// TIA Portal project "Hardware" (V14)

(* hardware
DEVICE "ET 200S-Station_1"  ET 200S station
   slot 0: "Baugruppenträger_0"  Rail
   slot 2: "PLC_1"  IM151-8 CPU  6ES7 151-8AB00-0AB0  V2.7
      slot 1: "PROFINET-Schnittstelle_1"  PN-IO
         slot 1: "Port_1"  Port
         slot 2: "Port_2"  Port
         slot 3: "Port_3"  Port
   slot 4: "PM-E 24VDC_1"  PM-E 24VDC  6ES7 138-4CA01-0AA0
   slot 5: "4AI x I 2WIRE ST_1"  4AI x I 2WIRE ST  6ES7 134-4GD00-0AB0
   slot 6: "2AO x U ST_1"  2AO x U ST  6ES7 135-4FB01-0AB0
   slot 7: "8DI x 24VDC_1"  8DI x 24VDC  6ES7 131-4BF00-0AA0
   slot 8: "8DI x 24VDC_2"  8DI x 24VDC  6ES7 131-4BF00-0AA0
   slot 9: "8DI x 24VDC_3"  8DI x 24VDC  6ES7 131-4BF00-0AA0
   slot 10: "8DI x 24VDC_4"  8DI x 24VDC  6ES7 131-4BF00-0AA0
   slot 11: "8DO x 24VDC / 0.5A_1"  8DO x 24VDC / 0.5A  6ES7 132-4BF00-0AA0
   slot 12: "8DO x 24VDC / 0.5A_2"  8DO x 24VDC / 0.5A  6ES7 132-4BF00-0AA0
   slot 13: "8DO x 24VDC / 0.5A_3"  8DO x 24VDC / 0.5A  6ES7 132-4BF00-0AA0
   slot 14: "8DO x 24VDC / 0.5A_4"  8DO x 24VDC / 0.5A  6ES7 132-4BF00-0AA0
DEVICE "HMI_1"  TP 177B 6'' PN/DP
   slot 0: "TP 177B 6'' PN/DP"  TP 177B 6'' PN/DP  6AV6 642-0BA01-1AX1  11.0.2.0
   slot 1: "HMI_RT_1"  TP 177B 6'' PN/DP  6AV6 642-0BA01-1AX1  11.0.2.0
   slot 5: "HMI_1.IE_CP_1"  PROFINET Interface  11.0.0.0
      slot 1: "PROFINET Schnittstelle_1"  PROFINET Interface
         slot 1: "Port_1"  Port
   slot 7: "HMI_1.MPI/DP_CP_1"  MPI/DP Interface  11.0.0.0
*)

// ===== PLC "PLC_1"  IM151-8 CPU =====

DATA_BLOCK "DB1"   // DB1
{ S7_Optimized_Access := 'FALSE' }
VERSION : 0.1
   VAR
      Static_0 : Int := 0;
      Static_1 : DInt := 0;
      Static_2 : Real := -1.0;
      Static_3 : Real := -1.0;
      Static_4 : Bool := FALSE;
   END_VAR
BEGIN
END_DATA_BLOCK

DATA_BLOCK "DB2"   // DB2
{ S7_Optimized_Access := 'FALSE' }
VERSION : 0.1
   VAR
      Static_0 : Int := 0;
      Static_1 : Array[0..2, 0..9] of Real;
      Static_2 : Real := 50.0;
      Static_3 : Real := 30.0;
      Static_4 : Real := 20.0;
      Static_5 : Bool := FALSE;
   END_VAR
BEGIN
   Static_1[0,0] := 50.0;
   Static_1[0,1] := 0.0;
   Static_1[0,2] := 0.0;
   Static_1[0,3] := 0.0;
   Static_1[0,4] := 0.0;
   Static_1[0,5] := 0.0;
   Static_1[0,6] := 0.0;
   Static_1[0,7] := 0.0;
   Static_1[0,8] := 0.0;
   Static_1[0,9] := 0.0;
   Static_1[1,0] := 30.0;
   Static_1[1,1] := 0.0;
   Static_1[1,2] := 0.0;
   Static_1[1,3] := 0.0;
   Static_1[1,4] := 0.0;
   Static_1[1,5] := 0.0;
   Static_1[1,6] := 0.0;
   Static_1[1,7] := 0.0;
   Static_1[1,8] := 0.0;
   Static_1[1,9] := 0.0;
   Static_1[2,0] := 20.0;
   Static_1[2,1] := 0.0;
   Static_1[2,2] := 0.0;
   Static_1[2,3] := 0.0;
   Static_1[2,4] := 0.0;
   Static_1[2,5] := 0.0;
   Static_1[2,6] := 0.0;
   Static_1[2,7] := 0.0;
   Static_1[2,8] := 0.0;
   Static_1[2,9] := 0.0;
END_DATA_BLOCK

DATA_BLOCK "DB3"   // DB3
{ S7_Optimized_Access := 'FALSE' }
VERSION : 0.1
   VAR
      Static_0 : Int := 0;
      Static_1 : Int := 0;
      Static_2 : Int := 0;
   END_VAR
BEGIN
END_DATA_BLOCK

DATA_BLOCK "DB100"   // DB100
{ S7_Optimized_Access := 'FALSE' }
VERSION : 0.1
   VAR
      Static_0 : Real := 0.0;
      Static_1 : Real := 0.0;
      Static_2 : Real := 0.0;
   END_VAR
BEGIN
END_DATA_BLOCK

DATA_BLOCK "DB101"   // DB101
{ S7_Optimized_Access := 'FALSE' }
VERSION : 0.1
   VAR
      Static_0 : Int := 0;
   END_VAR
BEGIN
END_DATA_BLOCK

FUNCTION "FC1" : Real   // FC1, FBD
{ S7_Optimized_Access := 'FALSE' }
VERSION : 0.1
   VAR_INPUT
      Input_0 : Int;
      Input_1 : DInt;
   END_VAR
   VAR_TEMP
      Temp_0 : DInt;
      Temp_1 : DInt;
      Temp_2 : DInt;
      Temp_3 : Real;
      Temp_4 : Real;
      Temp_5 : Real;
   END_VAR
BEGIN

REGION Network 1
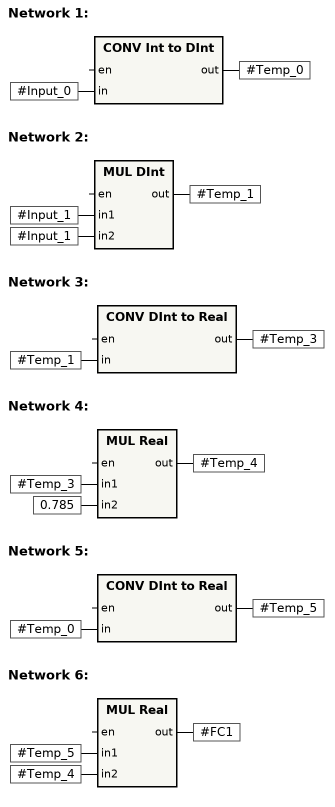
   #Temp_0 := INT_TO_DINT(#Input_0);
END_REGION

REGION Network 2
   #Temp_1 := #Input_1 * #Input_1;
END_REGION

REGION Network 3
   #Temp_3 := DINT_TO_REAL(#Temp_1);
END_REGION

REGION Network 4
   #Temp_4 := #Temp_3 * 0.785;
END_REGION

REGION Network 5
   #Temp_5 := DINT_TO_REAL(#Temp_0);
END_REGION

REGION Network 6
   #FC1 := #Temp_5 * #Temp_4;
END_REGION
END_FUNCTION

FUNCTION "FC2" : Real   // FC2, SCL
{ S7_Optimized_Access := 'FALSE' }
VERSION : 0.1
   VAR_INPUT
      Input_0 : Int;
      Input_1 : DInt;
   END_VAR
BEGIN
         SET;
         SAVE;
         =     %L0.0;
         L     #Input_0;
         L     0;
         >I;
         =     %L0.1;
         L     #Input_1;
         L     DINT#0;
         >D;
         A     %L0.1;
         JCN   M001;
         TAK;
         DTR;
         PUSH;
         *R;
         L     DINT#1_061_746_115;
         *R;
         T     %LD2;
         L     #Input_0;
         ITD;
         DTR;
         L     %LD2;
         *R;
         T     #FC2;
         JU    M002;
   M001: L     DINT#-1_082_130_432;
         T     #FC2;
   M002: CLR;
         A     %L0.0;
         SAVE;
END_FUNCTION

FUNCTION "FC3" : Real   // FC3, SCL
{ S7_Optimized_Access := 'FALSE' }
VERSION : 0.1
   VAR_INPUT
      Input_0 : Int;
   END_VAR
BEGIN
         SET;
         SAVE;
         =     %L0.0;
         L     #Input_0;
         L     -40;
         <I;
         =     %L0.1;
         TAK;
         L     -4800;
         >=I;
         A     %L0.1;
         JCN   M001;
         TAK;
         ITD;
         DTR;
         L     DINT#1_109_393_408;
         +R;
         L     DINT#-1_005_273_088;
         /R;
         T     #FC3;
         JU    M002;
   M001: L     DINT#-1_082_130_432;
         T     #FC3;
   M002: CLR;
         A     %L0.0;
         SAVE;
END_FUNCTION

FUNCTION "FC4" : Void   // FC4, SCL
{ S7_Optimized_Access := 'FALSE' }
VERSION : 0.1
   VAR_INPUT
      Input_0 : Bool;
      Input_1 : Int;
   END_VAR
   VAR_IN_OUT
      InOut_0 : Array[0..2, 0..9] of Real;
      InOut_1 : Real;
      InOut_2 : Real;
      InOut_3 : Real;
   END_VAR
BEGIN
         SET;
         SAVE;
         =     %L0.0;
         L     #Input_1;
         ITD;
         T     %LD2;
         L     DINT#32;
         *D;
         L;
         LAR1;
         TAK;
         L     W [ AR1 , P#0.0 ];
         T     %LW10;
         TAK;
         L     D [ AR1 , P#2.0 ];
         +D;
         T     %LD6;
         L     %LD2;
         L     DINT#10;
         +D;
         L     DINT#32;
         *D;
         L;
         LAR1;
         TAK;
         L     W [ AR1 , P#0.0 ];
         T     %LW16;
         TAK;
         L     D [ AR1 , P#2.0 ];
         +D;
         T     %LD12;
         L     %LD2;
         L     DINT#20;
         +D;
         L     DINT#32;
         *D;
         L;
         LAR1;
         TAK;
         L     W [ AR1 , P#0.0 ];
         T     %LW22;
         TAK;
         L     D [ AR1 , P#2.0 ];
         +D;
         T     %LD18;
         A     #Input_0;
         JCN   M001;
         L     #InOut_1;
         L     DINT#1_120_403_456;
         >R;
         JCN   M002;
         T     #InOut_1;
   M002: L     #InOut_1;
         OPN   DB [ %LW10 ];
         LAR1  %LD6;
         T     D [ AR1 , P#0.0 ];
         L     DINT#1_120_403_456;
         L     #InOut_1;
         -R;
         T     %LD2;
         L     #InOut_1;
         L     #InOut_2;
         +R;
         L     DINT#1_120_403_456;
         >R;
         JCN   M003;
         L     %LD2;
         T     #InOut_2;
   M003: L     #InOut_2;
         L     DINT#0;
         <R;
         JCN   M004;
         T     #InOut_2;
   M004: L     #InOut_2;
         OPN   DB [ %LW16 ];
         LAR1  %LD12;
         T     D [ AR1 , P#0.0 ];
         L     %LD2;
         L     #InOut_2;
         -R;
         T     #InOut_3;
         OPN   DB [ %LW22 ];
         LAR1  %LD18;
         T     D [ AR1 , P#0.0 ];
         JU    M005;
   M001: OPN   DB [ %LW10 ];
         LAR1  %LD6;
         L     D [ AR1 , P#0.0 ];
         T     #InOut_1;
         OPN   DB [ %LW16 ];
         LAR1  %LD12;
         L     D [ AR1 , P#0.0 ];
         T     #InOut_2;
         OPN   DB [ %LW22 ];
         LAR1  %LD18;
         L     D [ AR1 , P#0.0 ];
         T     #InOut_3;
   M005: CLR;
         A     %L0.0;
         SAVE;
END_FUNCTION

FUNCTION "FC5" : Real   // FC5, FBD
{ S7_Optimized_Access := 'FALSE' }
VERSION : 0.1
   VAR_INPUT
      Input_0 : Int;
      Input_1 : Int;
   END_VAR
   VAR_TEMP
      Temp_0 : DInt;
      Temp_1 : Real;
      Temp_2 : Int;
      Temp_3 : DInt;
      Temp_4 : Real;
      Temp_5 : Real;
      Temp_6 : Real;
   END_VAR
BEGIN

REGION Network 1
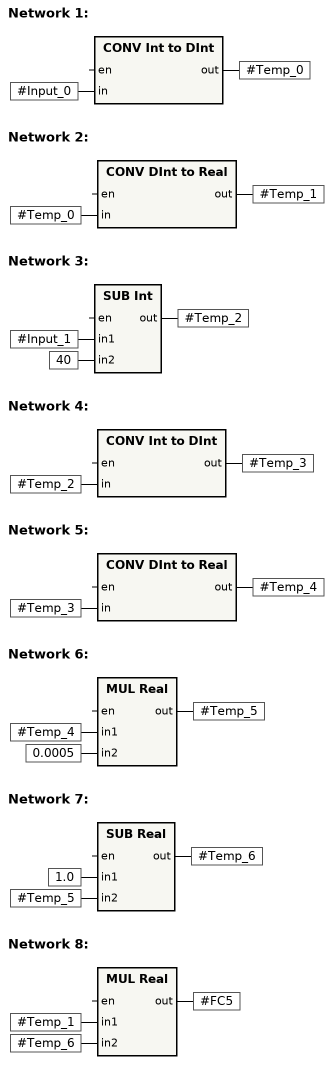
   #Temp_0 := INT_TO_DINT(#Input_0);
END_REGION

REGION Network 2
   #Temp_1 := DINT_TO_REAL(#Temp_0);
END_REGION

REGION Network 3
   #Temp_2 := #Input_1 - 40;
END_REGION

REGION Network 4
   #Temp_3 := INT_TO_DINT(#Temp_2);
END_REGION

REGION Network 5
   #Temp_4 := DINT_TO_REAL(#Temp_3);
END_REGION

REGION Network 6
   #Temp_5 := #Temp_4 * 0.0005;
END_REGION

REGION Network 7
   #Temp_6 := 1.0 - #Temp_5;
END_REGION

REGION Network 8
   #FC5 := #Temp_1 * #Temp_6;
END_REGION
END_FUNCTION

ORGANIZATION_BLOCK "OB1"   // OB1, FBD
{ S7_Optimized_Access := 'FALSE' }
VERSION : 0.1
   VAR_TEMP
      Temp_0 : Byte;
      Temp_1 : Byte;
      Temp_2 : Byte;
      Temp_3 : Byte;
      Temp_4 : Byte;
      Temp_5 : Byte;
      Temp_6 : Int;
      Temp_7 : Int;
      Temp_8 : Int;
      Temp_9 : Date_And_Time;
   END_VAR
BEGIN

REGION Network 1
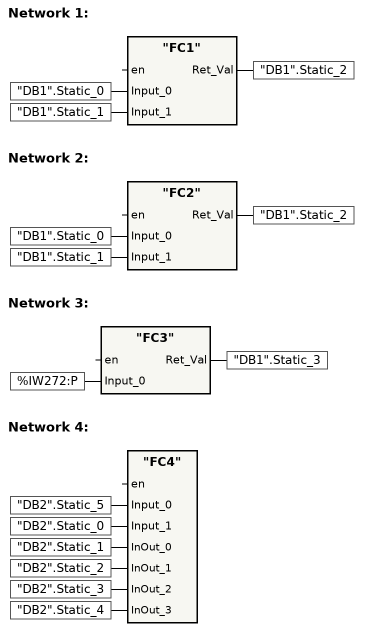
   "DB1".Static_2 := "FC1"(Input_0 := "DB1".Static_0, Input_1 := "DB1".Static_1);
END_REGION

REGION Network 2
   "DB1".Static_2 := "FC2"(Input_0 := "DB1".Static_0, Input_1 := "DB1".Static_1);
END_REGION

REGION Network 3
   "DB1".Static_3 := "FC3"(Input_0 := %IW272:P);
END_REGION

REGION Network 4
   "FC4"(Input_0 := "DB2".Static_5,
         Input_1 := "DB2".Static_0,
         InOut_0 := "DB2".Static_1,
         InOut_1 := "DB2".Static_2,
         InOut_2 := "DB2".Static_3,
         InOut_3 := "DB2".Static_4);
END_REGION
END_ORGANIZATION_BLOCK

(* ===== HMI "HMI_RT_1" =====
system functions are stored by id; their names below are inferred from use
connection "HMI_Verbindung_1": ETHERNET, SIMATIC S7 300/400 MPI
connection "HMI_Verbindung_2": ETHERNET, SIMATIC S7 300/400 MPI

HMI tags "Standard-Variablentabelle"
   "Variable_Bildnummer" : UInt, internal
   "A_rot" : Bool = PLC A_rot AT %A9.6, 1 s
   "A_gelb" : Bool = PLC A_gelb AT %A9.7, 1 s
   "A_gruen" : Bool = PLC A_gruen AT %A10.0, 1 s
   "FG_rot" : Bool = PLC FG_rot AT %A10.6, 1 s
   "FG_gruen" : Bool = PLC FG_gruen AT %A10.7, 1 s
   "Variable_Tag_S" : Int = PLC Variable.Tag_S AT %DB3.DBW4, 1 s
   "Variable_Tag_M" : Int = PLC Variable.Tag_M AT %DB3.DBW6, 1 s
   "Variable_Nacht_S" : Int = PLC Variable.Nacht_S AT %DB3.DBW10, 1 s
   "Variable_Nacht_M" : Int = PLC Variable.Nacht_M AT %DB3.DBW12, 1 s

text list "Textliste_Bildnamen": 1 'Grundbild'; 2 'Ampel'; 3 'Uhrzeit'

screen "Grundbild" 320x200, template "Vorlage_1"
   on GenerateScreen: SetTag("Variable_Bildnummer", 1)
   TextField "HmiScreenItemData" at 32,55 size 256x36; Text 'Willkommen zum HMI_1 (TP 177B 6″ PN/DP)!'
   Button "Ampel" at 1,1 size 104x36; TextOff 'Ampel'
      on Release: ActivateScreen("Ampel", 0)
   Button "Uhrzeit" at 105,1 size 104x36; TextOff 'Uhrzeit'
      on Release: ActivateScreen("Uhrzeit", 0)

Template "Vorlage_1" 320x200
   Button "Beenden" at 267,150 size 51x47; TextOff 'Beenden'; PictureOff "ExitRuntime_TP_177B_6_PNDP"; PictureOn "ExitRuntime_TP_177B_6_PNDP"
      on Release: StopRuntime(0)
   Button "Template_Button" at 214,150 size 51x47; TextOff 'Text'
   Button "Template_Button_1" at 160,150 size 51x47; TextOff 'Text'
   Button "Template_Button_2" at 107,150 size 51x47; TextOff 'Text'
   Button "Template_Button_3" at 54,150 size 51x47; TextOff 'Text'
   Button "Startbild" at 1,150 size 51x47; TextOff 'Startbild'; PictureOff "NavigateHome_TP_177B_6_PNDP"; PictureOn "NavigateHome_TP_177B_6_PNDP"
      on Release: ActivateScreen("Grundbild", 0)

screen "Ampel" 320x200, template "Vorlage_1"
   on GenerateScreen: SetTag("Variable_Bildnummer", 2)
   GraphicView "Grafikanzeige_1" at 0,1 size 318x150; Picture "strasse"
   Group "Group" at 167,1 size 80x32
   Group "Group_1" at 73,119 size 80x32
   Group "Group_2" at 112,1 size 26x43
   Group "Group_3" at 188,107 size 26x43
   Circle "Kreis_1" at 171,7 size 21x21
      Visibility <- "A_rot"
   Circle "Kreis_2" at 194,6 size 23x23
      Appearance <- "A_gelb"
   Circle "Kreis_3" at 219,6 size 26x26
      Appearance <- "A_gruen"
   Circle "Kreis_4" at 128,125 size 21x21
      Visibility <- "A_rot"
   Circle "Kreis_5" at 103,124 size 23x23
      Appearance <- "A_gelb"
   Circle "Kreis_6" at 75,124 size 26x26
      Appearance <- "A_gruen"
   Circle "Kreis_7" at 118,5 size 16x16
      Visibility <- "FG_rot"
   Circle "Kreis_8" at 118,24 size 16x16
      Appearance <- "FG_gruen"
   Circle "Kreis_9" at 192,130 size 16x16
      Visibility <- "FG_rot"
   Circle "Kreis_10" at 192,111 size 16x16
      Appearance <- "FG_gruen"

screen "Uhrzeit" 320x200, template "Vorlage_1"
   on GenerateScreen: SetTag("Variable_Bildnummer", 3)
   Button "Zurück" at 1,1 size 104x36; TextOff 'Zurück'
      on Release: ActivateScreen("Grundbild", 0)
   TextField "Textfeld_1" at 38,63 size 31x20; Text 'Tag:'
   IOField "EA-Feld_1" at 69,64 size 29x20; FormatPattern 99
      ProcessValue <- "Variable_Tag_S"
   TextField "Textfeld_2" at 97,64 size 10x20; Text ':'
   IOField "EA-Feld_2" at 107,64 size 24x20; FormatPattern 99
      ProcessValue <- "Variable_Tag_M"
   TextField "Textfeld_3" at 134,65 size 24x20; Text 'Uhr'
   TextField "Textfeld_4" at 28,98 size 41x20; Text 'Nacht:'
   IOField "EA-Feld_3" at 68,100 size 29x20; FormatPattern 99
      ProcessValue <- "Variable_Nacht_S"
   TextField "Textfeld_5" at 97,100 size 10x20; Text ':'
   IOField "EA-Feld_4" at 107,100 size 24x20; FormatPattern 99
      ProcessValue <- "Variable_Nacht_M"
   TextField "Textfeld_6" at 133,101 size 24x20; Text 'Uhr'
*)